// TIA Portal V17 export
// export: Created 2024-08-07T21:44:10.0241445Z, ExportSetting WithDefaults, DisplayName Totally Integrated Automation Portal, DisplayVersion V17 Update 7, DisplayName TIA Portal Openness, DisplayVersion V17 Update 7, DisplayName TIA Portal Version Control Interface, DisplayVersion V17, DisplayName SINAMICS Startdrive Advanced, DisplayVersion V17 SP2, DisplayName SINAMICS Startdrive G110M, G120, G120C, G120D, G120P, G115D, DisplayVersion V17 SP2, DisplayName SINAMICS Startdrive G130, G150, S120, S150, SINAMICS MV, S210, DisplayVersion V17 SP2, DisplayName STEP 7 Professional, DisplayVersion V17 Update 7, DisplayName STEP 7 Safety, DisplayVersion V17 Update 6, DisplayName WinCC Advanced / Unified PC, DisplayVersion V17 Update 7
FUNCTION "Extract_data_DMC" : Void   // FC2011, LAD
{ S7_Optimized_Access := 'TRUE' }
VERSION : 0.1
// stored: AutoNumber false, IsIECCheckEnabled false, SetENOAutomatically false, UDAEnableTagReadback false
   VAR_INPUT
      round : Byte;
      Data_DMC : Array[1.."MaxRoundNumber", 1..10] of "DATA_DMC";
   END_VAR
   VAR_OUTPUT
      DATA_DMC_Extract : Array[1..10] of String[25];
   END_VAR
   VAR_TEMP
      idx : SInt;
      round_idx : SInt;
   END_VAR
BEGIN

REGION Network 1
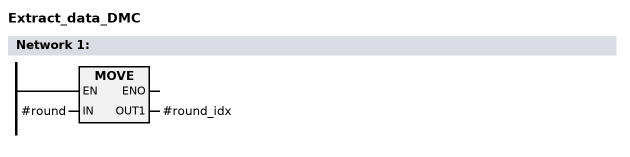
   RUNG wire#powerrail
      Move(in := #round, out1 => #round_idx)
   END_RUNG
   // the same network as SCL:
   #round_idx := #round;
END_REGION

REGION Network 2 (SCL)
   FOR  #idx:=1 TO 10 DO
       #DATA_DMC_Extract[#idx]:= #Data_DMC[#round_idx,#idx].SAP_REF_PRODUCTION;

   END_FOR;
END_REGION
END_FUNCTION
